FUNCTION_BLOCK PUBLISH_3 (* Three-Variable Publisher *)
  (* Standard: 61499-1-F.2.1; Classification: Communications; Function: PUBLISH *)
  (* Version 0.0, 2001-04-27, JHC, Rockwell Automation, XML version *)
  (* Version 0.0, 1998-12-08, JHC, Rockwell Automation, SRC version *)
  (* Compiler header: package fb.rt.net; *)
  (* Compiler Java IBM VisualAge 3.0 *)
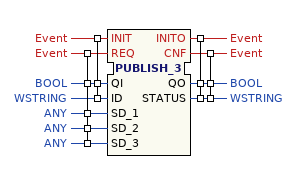
  EVENT_INPUT
    INIT WITH QI, ID; (* Service Initialization *)
    REQ WITH QI, SD_1, SD_2, SD_3; (* Service Request *)
  END_EVENT
  EVENT_OUTPUT
    INITO WITH QO, STATUS; (* Initialization Confirm *)
    CNF WITH QO, STATUS; (* Service Confirmation *)
  END_EVENT
  VAR_INPUT
    QI : BOOL; (* Event Input Qualifier *)
    ID : WSTRING; (* Connection Identifier *)
    SD_1 : ANY; (* Data to Send *)
    SD_2 : ANY; (* Data to Send *)
    SD_3 : ANY; (* Data to Send *)
  END_VAR
  VAR_OUTPUT
    QO : BOOL; (* Event Output Qualifier *)
    STATUS : WSTRING; (* Service Status *)
  END_VAR
  SERVICE PUBLISH_3/SUBSCRIBE_3 (* Data Publication Service *)
    SEQUENCE normal_establishment
      PUBLISH_3.INIT+(ID) -> PUBLISH_3.INITO+();
      SUBSCRIBE_3.INIT+(ID) -> SUBSCRIBE_3.INITO+();
    END_SEQUENCE
    SEQUENCE publisher_rejected_establishment
      PUBLISH_3.INIT+(ID) -> PUBLISH_3.INITO-(STATUS);
    END_SEQUENCE
    SEQUENCE subscriber_rejected_establishment
      SUBSCRIBE_3.INIT+(ID) -> SUBSCRIBE_3.INITO-(STATUS);
    END_SEQUENCE
    SEQUENCE normal_data_transfer
      PUBLISH_3.REQ+(SD_1,SD_2,SD_3) -> SUBSCRIBE_3.IND+(RD_1,RD_2,RD_3);
      -> PUBLISH_3.CNF+();
      SUBSCRIBE_3.RSP+();
    END_SEQUENCE
    SEQUENCE data_transfer_error
      PUBLISH_3.REQ+(SD_1,SD_2,SD_3) -> SUBSCRIBE_3.IND-(STATUS);
      -> PUBLISH_3.CNF+();
    END_SEQUENCE
    SEQUENCE publisher_initiated_disconnect
      PUBLISH_3.INIT-() -> SUBSCRIBE_3.INITO-(STATUS);
      -> PUBLISH_3.INITO-(STATUS);
    END_SEQUENCE
    SEQUENCE subscriber_initiated_disconnect
      SUBSCRIBE_3.INIT-() -> SUBSCRIBE_3.INITO-(STATUS);
    END_SEQUENCE
    SEQUENCE system_publisher_disconnect
      -> PUBLISH_3.INITO-(STATUS);
      -> SUBSCRIBE_3.INITO-(STATUS);
    END_SEQUENCE
    SEQUENCE system_subscriber_disconnect
      -> SUBSCRIBE_3.INITO-(STATUS);
    END_SEQUENCE
  END_SERVICE
END_FUNCTION_BLOCK
